(* CODESYS project OPCUA-server.project

Project tree, tasks and I/O mapping:
  Device : CODESYS Control Win V3, 3S - Smart Software Solutions GmbH, order no. 305021, version 3.5.11.30
    application Application
      libraries: Standard, * (System)
      task MainTask (cyclic, interval t#20ms, priority 1) calls PLC_PRG
      program PLC_PRG [LD]
      Symbols
      function block Hours_Counter [ST]
    Ethernet : Ethernet, 3S - Smart Software Solutions GmbH, version 3.5.11.0
      ModbusTCP_Slave_Device : ModbusTCP Slave Device, 3S - Smart Software Solutions GmbH, version 3.5.11.0
          settings: Unit-ID = 3; StartAdresses.Coils = 2; StartAdresses.DiscreteInputs = 2; StartAdresses.HoldingRegister = 2; StartAdresses.InputRegister = 2; Data Model Options = 1
          input  Application.PLC_PRG.TON_0.Q : BOOL  // Inputs.Inputs.Bit0
          output Application.PLC_PRG.TON_0.Q : BOOL  // Outputs.Outputs.Bit0
          unmapped channels: Inputs, Outputs
*)

// Device/Application/PLC_PRG
PROGRAM PLC_PRG
VAR
	// Variáveis de controle
	Start: BOOL;
	Stop: BOOL;
	Ciclo: BOOL;
	Stop_Blade: BOOL;
	Reset: BOOL;
	Reset_Counter: BOOL;

	// Trigger de borda de subida
	R_TRIG_0: R_TRIG;

	// Variáveis relacionadas ao motor
	RPM_M1: INT;
	RPM_M2: INT;
	Corrente_M1: INT;
	Corrente_M2: INT;
	motor_feedback: BOOL;
	motor1_alert: BOOL;
	motor1_running: BOOL;

	// Variáveis relacionadas ao buffer
	Buffer_Conveyor: LREAL;
	Exit_Conveyor: LREAL;
	Buffer_Entry: WORD;
	Buffer_Exit: WORD;
	S_Buffer_Entry: BOOL;
	S_Buffer_Exit: BOOL;

	// Contadores IEC
	IEC_Counter_0_DB: CTU;
	IEC_Counter_0_DB_1: CTU;
	IEC_Counter_0_DB_2: CTU;

	// Sinal de saída
	S_Exit: BOOL;
	Exit_var: WORD;

	// Outras variáveis
	val: UINT;
	Sec: INT;
	Minutes: INT;
	Hours: INT;

	// Temporizadores e relógio
	TON_0: TON;
	Clock: TIME;
	TON_1: TON;
	Hours_Counter_0: Hours_Counter;
	oscilador: BOOL;

	// Variáveis de leitura
	Read_M1: BOOL;

	// Variáveis auxiliares
	var1: BOOL;
	var2: INT;
	var3: INT;

END_VAR
VAR // added by the converter: edge detectors and wires of the graphical bodies
    _w1, _w2, _w3 : BOOL;
END_VAR

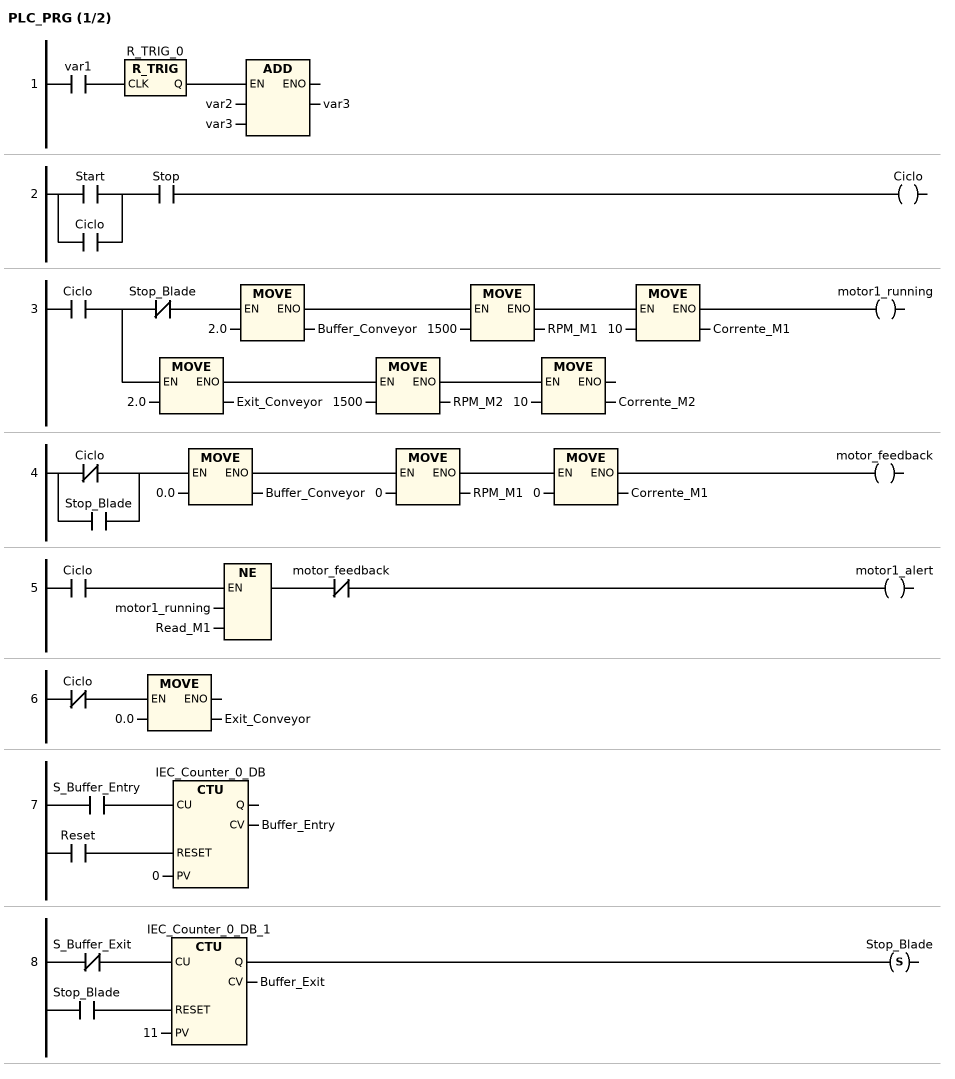
// NETWORK 1
R_TRIG_0(CLK := var1); // R_TRIG
IF R_TRIG_0.Q THEN var3 := var2 + var3; END_IF

// NETWORK 2
Ciclo := (Start OR Ciclo) AND Stop;

// NETWORK 3
_w1 := Ciclo AND NOT Stop_Blade;
IF _w1 THEN Buffer_Conveyor := 2.0; END_IF
IF _w1 THEN RPM_M1 := 1500; END_IF
IF _w1 THEN Corrente_M1 := 10; END_IF
motor1_running := _w1;
_w2 := Ciclo;
IF _w2 THEN Exit_Conveyor := 2.0; END_IF
IF _w2 THEN RPM_M2 := 1500; END_IF
IF _w2 THEN Corrente_M2 := 10; END_IF

// NETWORK 4
_w3 := NOT Ciclo OR Stop_Blade;
IF _w3 THEN Buffer_Conveyor := 0.0; END_IF
IF _w3 THEN RPM_M1 := 0; END_IF
IF _w3 THEN Corrente_M1 := 0; END_IF
motor_feedback := _w3;

// NETWORK 5
motor1_alert := (Ciclo AND motor1_running <> Read_M1) AND NOT motor_feedback;

// NETWORK 6
IF NOT Ciclo THEN Exit_Conveyor := 0.0; END_IF

// NETWORK 7
IEC_Counter_0_DB(CU := S_Buffer_Entry, RESET := Reset, PV := 0, CV => Buffer_Entry); // CTU

// NETWORK 8
IEC_Counter_0_DB_1(CU := NOT S_Buffer_Exit, RESET := Stop_Blade, PV := 11, CV => Buffer_Exit); // CTU
Stop_Blade S= IEC_Counter_0_DB_1.Q;

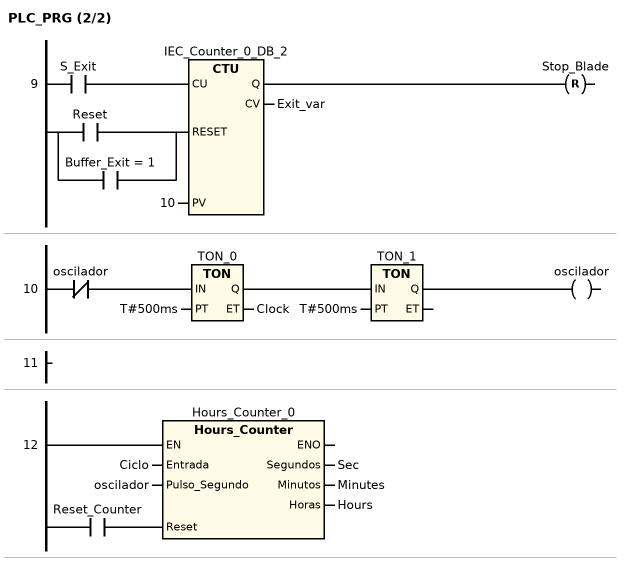
// NETWORK 9
IEC_Counter_0_DB_2(CU := S_Exit, RESET := Reset OR (Buffer_Exit = 1), PV := 10, CV => Exit_var); // CTU
Stop_Blade R= IEC_Counter_0_DB_2.Q;

// NETWORK 10
TON_0(IN := NOT oscilador, PT := T#500ms, ET => Clock); // TON
TON_1(IN := TON_0.Q, PT := T#500ms); // TON
oscilador := TON_1.Q;

// NETWORK 11

// NETWORK 12
Hours_Counter_0(
    Entrada := Ciclo,
    Pulso_Segundo := oscilador,
    Reset := Reset_Counter,
    Segundos => Sec,
    Minutos => Minutes,
    Horas => Hours); // Hours_Counter

END_PROGRAM

// Device/Application/Hours_Counter
FUNCTION_BLOCK Hours_Counter
VAR_INPUT
    Entrada : BOOL;
    Pulso_Segundo : BOOL;
    Reset : BOOL;
END_VAR

VAR_OUTPUT
	Segundos : INT;
    Minutos : INT;
    Horas : INT;
END_VAR

VAR
    
END_VAR

IF Entrada THEN
    IF Pulso_Segundo THEN
        Segundos := Segundos + 1;
        IF Segundos >= 60 THEN
            Segundos := 0;
            Minutos := Minutos + 1;
            IF Minutos >= 60 THEN
                Minutos := 0;
                Horas := Horas + 1;
            END_IF;
        END_IF;
    END_IF;
END_IF;

IF Reset THEN
    Segundos := 0;
    Minutos := 0;
    Horas := 0;
END_IF;

END_FUNCTION_BLOCK
